# EPICS IOC start-up script: ipApp/iocsh/MicroE_SS350.iocsh
#- ###################################################
#- PREFIX         - IOC Prefix
#- INSTANCE       - Instance Prefix
#- PORT           - Serial port name
#- IP             - Location of IP module
#- ###################################################

iocshLoad("$(IP)/iocsh/setSerialParams.iocsh", "PORT=$(PORT), BAUD=38400, BITS=8, STOP=1, PARITY=even")

dbLoadRecords("$(IP)/db/MicroE_SS350.vdb","P=$(PREFIX),N=$(INSTANCE),PORT=$(PORT)")
